{attribute 'pack_mode' := '2'}
TYPE ST_AXIS_MOVE_DATA :
STRUCT
  rSetPos           : LREAL;
  rSetVelo          : LREAL;
  rOverride         : LREAL := 100.0;
  rAcc              : LREAL;
  rDec              : LREAL;
  rJerk             : LREAL;
  iDirection        : INT;
END_STRUCT
END_TYPE

(* stored: Version 1.1.0.1, ProductVersion 3.1.4026.19
   DUT ST_AXIS_MOVE_DATA: Id {ca43e1e3-6fd4-0448-2567-b8eb25d99c7e} *)
